// TIA Portal V20 export
DATA_BLOCK "DataFromSafety"   // DB127
// stored: Access Published, AssignedProDiagFB Safety.ProDiag, InstanceOfName Safety.typeDataFromSafety, InstanceOfType UDT, Namespace Safety
"Safety.typeDataFromSafety"
   // VAR
   //    devicesSummary { ExternalWritable := 'False'} : "Safety.typeDevicesStatusSummary";
   //    mainOp { ExternalWritable := 'False'} : "Safety.typeMainOpMode";
   //    pHmi { ExternalWritable := 'False'} : "Safety.typePhmi";
   //    scsMode { ExternalWritable := 'False'} : "Safety.typeScsMode";
   //    rcMode1 { ExternalWritable := 'False'} : "Safety.typeRollChangeMode";
   //    rcMode2 { ExternalWritable := 'False'} : "Safety.typeRollChangeMode";
   //    scrapBox1 { ExternalWritable := 'False'} : "Safety.typeScrapBoxCommands";
   //    eStopStatus { ExternalWritable := 'False'} : "Safety.typeEstopStatus";
   //    fDoorSwitchStatus { ExternalWritable := 'False'} : "Safety.typeFDoorSwitchStatus";
   //    fDoorCoilStatus { ExternalWritable := 'False'} : "Safety.typeFDoorUnlockOutput";
   //    Zone1SafetyOpEnable { ExternalWritable := 'False'} : "Safety.typeSafetyOperationEnable";
   //    Zone2SafetyOpEnable { ExternalWritable := 'False'} : "Safety.typeSafetyOperationEnable";
   //    Zone3SafetyOpEnable { ExternalWritable := 'False'} : "Safety.typeSafetyOperationEnable";
   //    eStopZone1 { ExternalWritable := 'False'} : "Safety.typeEstopFunction";
   //    eStopZone2 { ExternalWritable := 'False'} : "Safety.typeEstopFunction";
   //    eStopZone3 { ExternalWritable := 'False'} : "Safety.typeEstopFunction";
   //    statusZone1 { ExternalWritable := 'False'} : "Safety.typeSafetyZoneStatus";
   //    statusZone2 { ExternalWritable := 'False'} : "Safety.typeSafetyZoneStatus";
   //    statusZone3 { ExternalWritable := 'False'} : "Safety.typeSafetyZoneStatus";
   //    fDoorDrive { ExternalWritable := 'False'} : "Safety.typeFDoorFunction";
   //    driveStatus { ExternalWritable := 'False'} : "Safety.typeSafetyDriveStatus";
   //    safetySensor { ExternalWritable := 'False'} : "Safety.typeSafetySensor";
   //    feedbackFault { ExternalWritable := 'False'} : "Safety.typeFeedbackFault";
   //    radiusStatus { ExternalWritable := 'False'} : "Safety.typeRadiusStatusSummary";
   //    cvCoverStatus { ExternalWritable := 'False'} : "Safety.typeCvCoverStatus";
   //    EnableACK { ExternalWritable := 'False'} : Bool;
   //    SS1Extention { ExternalWritable := 'False'} : Bool;
   //    LHSS1Extenstion { ExternalWritable := 'False'} : Bool;
   //    RHSS1Extenstion { ExternalWritable := 'False'} : Bool;
   //    AllEstopsOK { ExternalWritable := 'False'} : Bool;
   //    Z_Fold_AllEstopsOK { ExternalWritable := 'False'} : Bool;
   //    AllFdoorClose { ExternalWritable := 'False'} : Bool;
   //    AllSFDoorOpen { ExternalWritable := 'False'} : Bool;
   //    AnyNoMFDoorOpen { ExternalWritable := 'False'} : Bool;
   //    safetyReleasedAllSafetyZones { ExternalWritable := 'False'} : Bool;   // All safety zones are released OFF
   //    ackRequiredAnySafetyZone { ExternalWritable := 'False'} : Bool;
   //    ackOP_changeRequired { ExternalWritable := 'False'} : Bool;
   //    ackOperatorControlCondition { ExternalWritable := 'False'} : Bool;
   //    doorBoxAllReset { ExternalWritable := 'False'} : Bool;
   //    totalSafetyReset { ExternalWritable := 'False'} : Bool;
   //    zone1DoorOpenRequest { ExternalWritable := 'False'} : Bool;
   //    zone2DoorOpenRequest { ExternalWritable := 'False'} : Bool;
   //    zone3DoorOpenRequest { ExternalWritable := 'False'} : Bool;
   //    zone1DriveAckReq { ExternalWritable := 'False'} : Bool;
   //    zone2DriveAckReq { ExternalWritable := 'False'} : Bool;
   //    zone3DriveAckReq { ExternalWritable := 'False'} : Bool;
   //    noSafetyFault { ExternalWritable := 'False'} : Bool;
   //    connectionBoxID { ExternalWritable := 'False'} : Int;
   //    no_Corver_RC { ExternalWritable := 'False'} : Bool;
   //    LH_RollChangeActive { ExternalWritable := 'False'} : Bool;   // LH_Roll Change Active
   //    RH_RollChangeActive { ExternalWritable := 'False'} : Bool;   // RH_Roll Change Active
   //    FrameCoverNG { ExternalWritable := 'False'} : Bool;
   //    BA30CathodeCoverClose { ExternalAccessible := 'False'; ExternalVisible := 'False'; ExternalWritable := 'False'} : Bool;
   //    BA30AnodeCoverClose { ExternalAccessible := 'False'; ExternalVisible := 'False'; ExternalWritable := 'False'} : Bool;
   //    BA40CathodeCoverClose { ExternalAccessible := 'False'; ExternalVisible := 'False'; ExternalWritable := 'False'} : Bool;
   //    BA40AnodeCoverClose { ExternalAccessible := 'False'; ExternalVisible := 'False'; ExternalWritable := 'False'} : Bool;
   //    BA60ExternalDoorOpen { ExternalAccessible := 'False'; ExternalVisible := 'False'; ExternalWritable := 'False'} : Bool;
   //    BA60jrPPLeftDoorForcedOpen { ExternalAccessible := 'False'; ExternalVisible := 'False'; ExternalWritable := 'False'} : Bool;
   //    BA60jrPPLeftDoorNormalOpen { ExternalAccessible := 'False'; ExternalVisible := 'False'; ExternalWritable := 'False'} : Bool;
   //    BA60Stacker1LightCurtainDetect : Bool;
   //    BA60Stacker2LightCurtainDetect { ExternalAccessible := 'False'; ExternalVisible := 'False'; ExternalWritable := 'False'} : Bool;
   //    BA60Stacker2MaintanceDoorNormalOpen { ExternalAccessible := 'False'; ExternalVisible := 'False'; ExternalWritable := 'False'} : Bool;
   //    BA60Stacker2MaintanceDoorForcedOpen { ExternalAccessible := 'False'; ExternalVisible := 'False'; ExternalWritable := 'False'} : Bool;
   //    FdoorLamp : "Safety.fDoorLamp";
   //    DoorBoxUnlockSW : "Safety.typeDoorUnlockSW";
   //    BA015 { ExternalWritable := 'False'} : "Safety.s_PLC_Interlocks";
   //    BA030 { ExternalWritable := 'False'} : "Safety.s_PLC_Interlocks";
   //    BA040 { ExternalWritable := 'False'} : "Safety.s_PLC_Interlocks";
   //    BA060 { ExternalWritable := 'False'} : "Safety.s_PLC_Interlocks";
   // END_VAR
BEGIN
   // statusZone1.ackReq : Safety Zone 1 : Acknowledge oder Clear erforderlich
END_DATA_BLOCK
